(* IEC 61131-3 sources: IODBLib/, 7 files *)

(* ---- IODBLib.typ ---- *)
(********************************************************************
 * COPYRIGHT -- ARG
 ********************************************************************
 * Library: IODatabase
 * File: IODatabase.typ
 * Author: Administrator
 * Created: June 17, 2011
 ********************************************************************
 * Data types of library IODatabase
 ********************************************************************)

TYPE
	IODataBase : 	STRUCT
		Buffer : REFERENCE TO UDINT; (*Pointer to the allocated memory*)
		BufferSize : UDINT; (*size of the allocated memory*)
		DataTypeSize : UDINT; (*size of IODatapoint type*)
		ListDP : AsIOListDP; (*function block to get the IO on the system*)
		PVInfo : AsIOPVInfo; (*function block to get the PV's connected to the IO on the system*)
		State : USINT;
		NumberVariables : UINT;
	END_STRUCT;
	IODataPoint : 	STRUCT  (*DO NOT CHANGE ORDER: PVName, IODPType, INAName, IODPName*)
		PVName : STRING[80]; (*Name of the connected process variable*)
		IODPType : STRING[20]; (*Type of IO Point that is connected*)
		INAName : STRING[80]; (*INA address to slice*)
		IODPName : STRING[80]; (*Name of the connected IO datapoint*)
	END_STRUCT;
	Task_typ : 	STRUCT
		Name : STRING[80];
		Ident : UDINT;
		Group : USINT;
		State : USINT;
		Resource : SINT;
	END_STRUCT;
END_TYPE

(* ---- CreateIODatabase.st ---- *)
(********************************************************************
 * COPYRIGHT -- ARG
 ********************************************************************
 * Library: IODatabase
 * File: InitIODatabase.st
 * Author: Josh Polansky
 * Created: June 17, 2011
 ********************************************************************
 * Implementation of library IODatabase
 ********************************************************************)

//This MUST be called in INIT and must finish before calling GetINAInfo()

//Goes through all the IO and finds the number of connected datapoints

//Allocates memory

//Fills memory with datapoint info

FUNCTION CreateIODB

//Set return value to get rid of compiler warning

CreateIODB:=	0;

FOR iteration:= 0 TO 5 DO
	CASE Database.State OF

		1://Init
			Database.NumberVariables:=0;
			Database.ListDP.pLastDatapoint:= 0;
			Database.ListDP.enable:=1;
			Database.ListDP();
			IF Database.ListDP.status = 0 THEN
			  	Database.State:= 	2;
			END_IF

		2://We have a datapoint!
			IF Database.ListDP.pDatapoint <> 0
				THEN
			  	Database.State := 				3;
				Database.PVInfo.index:=			0;
				Database.PVInfo.pDatapoint:=	Database.ListDP.pDatapoint;
				Database.PVInfo.enable:=		1;
				Database.PVInfo();
				TempString ACCESS Database.PVInfo.pDatapoint;
			ELSE
			  	Database.State := 	0;
				CreateIODB:=		1;
			END_IF

		3://Get the status

			Database.PVInfo();

			IF Database.PVInfo.status = 0 //We have the info
				THEN
			  	Database.State := 	4;
			ELSIF Database.PVInfo.status = ERR_FUB_BUSY //We are getting the info
				THEN

			ELSE	//We couldn't get info, get the next one
			  	Database.State := 	5;
			END_IF

		4://Parse
			IF Database.PVInfo.pPvName <> 0 THEN

				//Get the current place in the buffer
				DataPoint  ACCESS (Database.Buffer + (Database.NumberVariables * Database.DataTypeSize));

				//Set the PV Name
				TempString ACCESS Database.PVInfo.pPvName;
				DataPoint.PVName:=	TempString;

				//Set the IO Datapoint name
				TempString ACCESS Database.ListDP.pDatapoint;
				DataPoint.IODPName:=	TempString;

				//Get the IO Type
				strind:=0;
				Done:=0;
				WHILE strind < brsstrlen(Database.ListDP.pDatapoint)
					AND strind < SIZEOF(DataPoint.IODPType)
					AND NOT Done
					DO
					IF	brsmemcmp( Database.ListDP.pDatapoint + strind,ADR('.'),1) = 0
					OR	brsmemcmp( Database.ListDP.pDatapoint + strind,ADR(':'),1) = 0
						THEN
						brsstrcpy( ADR(DataPoint.IODPType), Database.ListDP.pDatapoint );
						brsmemset( ADR(DataPoint.IODPType) + strind, 0, SIZEOF(DataPoint.IODPType)- strind);
						brsstrcpy( ADR(DataPoint.INAName),  Database.ListDP.pDatapoint + strind + 1 );
						Done:=1;
					END_IF
					strind:=strind+1;
				END_WHILE;

				len:= UDINT_TO_INT(brsstrlen( ADR(DataPoint.INAName) ));
				Done:=0;
				//Start at the end and look for the last "." to separate the INA device from the IODatapoint name
				WHILE( len > 0 AND NOT Done )  DO
					IF ( brsmemcmp( ADR(DataPoint.INAName) + len - 1, ADR('.' ), 1 ) = 0 )THEN
						Done := 1;
					END_IF
					TempString ACCESS ADR(DataPoint.INAName) + len - 1;
					len := len - 1;
				END_WHILE;

				brsstrcpy(ADR(DataPoint.IODPName),ADR(TempString)+1);
				TempString := '';

				Database.NumberVariables:= Database.NumberVariables+1;
				Database.State:= 	3;
				Database.PVInfo.index:=	Database.PVInfo.index+1;
			ELSE

				IF Database.PVInfo.index = 0 THEN
					Database.PVInfo.index:=	1;
					Database.State:= 	3;
				ELSE
					Database.State:= 	5;
				END_IF
			END_IF

		5://Get the next one
			Database.ListDP.pLastDatapoint:= Database.ListDP.pDatapoint;
			Database.ListDP();
			IF Database.ListDP.status = 0
				THEN
			  	Database.State:= 	2;
			ELSIF Database.ListDP.pDatapoint = 0 THEN
				Database.State := 	0;
			END_IF

	END_CASE;
END_FOR

END_FUNCTION

(* ---- GetChannelNum.st ---- *)
(********************************************************************
 * COPYRIGHT --
 ********************************************************************
 * Library: DPLookup
 * File: GetChannelNum.st
 * Author: Josh
 * Created: November 12, 2012
 ********************************************************************
 * Implementation of library DPLookup
 ********************************************************************)

(*  *)
FUNCTION GetChannelNum

	pDatapoint ACCESS GetINAInfo(DataBase,Datapoint,DPName);

	IF ADR(pDatapoint) <> 0 THEN
		DPName:=RIGHT(pDatapoint.IODPName,2);
		GetChannelNum := brsatoi( ADR(DPName));
	END_IF

END_FUNCTION

(* ---- GetINAInfo.st ---- *)
(********************************************************************
 * COPYRIGHT -- ARG
 ********************************************************************
 * Library: IODatabase
 * File: GetINAInfo.st
 * Author: Josh Polansky
 * Created: June 20, 2011
 ********************************************************************
 * Implementation of library IODatabase
 ********************************************************************)

FUNCTION GetINAInfo

(****************************************)
(* Check for invalid database 			*)
(****************************************)

IF( DataBase.Buffer = 0 )THEN

	GetINAInfo:=	0;
	INADeviceName:=	'Database not initialized';

	RETURN;

END_IF

(****************************************************************************)
(* Search through database for a PVName which matches the Datapoint input	*)
(****************************************************************************)

pDatapoint ACCESS (DataBase.Buffer + (DataBase.DataTypeSize * index) );

WHILE pDatapoint.PVName <> Datapoint AND index < DataBase.BufferSize/ DataBase.DataTypeSize DO

	pDatapoint ACCESS (DataBase.Buffer + (DataBase.DataTypeSize * index) );
	index:= index+1;

END_WHILE;

(****************************************)
(* Set return value						*)
(****************************************)

IF pDatapoint.PVName = Datapoint THEN

	GetINAInfo:=	ADR(pDatapoint);
	INADeviceName:=	pDatapoint.INAName;

ELSE

	GetINAInfo:=	0;
	INADeviceName:=	'Datapoint not found';

END_IF

END_FUNCTION

(* ---- InitIODatabase.st ---- *)
(*
 * File: InitIODatabase.st
 * Copyright (c) 2023 Loupe
 * https://loupe.team
 *
 * This file is part of IODBLib, licensed under the MIT License.
 *)

//This MUST be called in INIT and must finish before calling GetINAInfo()

//Goes through all the IO and finds the number of connected datapoints

//Allocates memory

//Fills memory with datapoint info

FUNCTION InitIODB

//Set return value to get rid of compiler warning

InitIODB:=	0;

//Get size of required buffer

Database.Buffer:=		0;
Database.BufferSize:=	0;
Database.DataTypeSize:=	SIZEOF( DataPoint);

//Get the first IO datapoint

Database.ListDP.pLastDatapoint:=	0;
Database.ListDP.enable:=			1;
Database.ListDP();

//Go through all the datapoints IO datapoints and check to see if they are connected to a PV datapoint

WHILE Database.ListDP.pDatapoint <> 0 // 0 means no datapoint was found
	DO

	Database.ListDP.pLastDatapoint:= Database.ListDP.pDatapoint;
	Database.ListDP();

	//If the status is 0 a datapoint was found

	IF ( Database.ListDP.status = 0 ) THEN

		//If we found a datapoint, check if it is connected to a PV

		Database.PVInfo.pDatapoint:=	Database.ListDP.pDatapoint;
		Database.PVInfo.enable:=		1;
		Database.PVInfo.index:=0;
		Database.PVInfo();
		IF Database.PVInfo.pDatapoint <> 0 THEN
			TempString ACCESS Database.PVInfo.pDatapoint;
//			logError('IOFound',TempString);
		END_IF

		//If there is a PV connected, add the size of the PV info to the buffer size

		//Get the producer
		IF Database.PVInfo.pPvName <> 0 THEN
			TempString ACCESS Database.PVInfo.pPvName;
//			logError('ProdPVFound',TempString);
			Database.BufferSize:= Database.BufferSize + Database.DataTypeSize;
		END_IF;

		Database.PVInfo.index:= Database.PVInfo.index+1;
		Database.PVInfo();

		//Get the Consumers
		WHILE Database.PVInfo.pPvName <> 0 DO
			TempString ACCESS Database.PVInfo.pPvName;
//			logError('ConsPVFound',TempString);
			Database.BufferSize:= Database.BufferSize + Database.DataTypeSize;
			Database.PVInfo.index:= Database.PVInfo.index+1;
			Database.PVInfo();
		END_WHILE;

	END_IF

END_WHILE;

//Get buffer

IF ( TMP_alloc(	Database.BufferSize,ADR(Database.Buffer)) = 0 )THEN
	Database.State:=1;
END_IF

END_FUNCTION

(* ---- GetTaskInfo.st ---- *)
(*
 * File: GetTaskInfo.st
 * Copyright (c) 2023 Loupe
 * https://loupe.team
 *
 * This file is part of IODBLib, licensed under the MIT License.
 *)

(*  *)
FUNCTION_BLOCK GetTaskInfo

	CASE State OF
		0:
			Status:= ERR_FUB_BUSY;
			IF ST_name(0,ADR(Info.Name),ADR(Info.Group)) = 0 THEN
				State:=1;
			END_IF

		1:
			IF ST_ident(ADR(Info.Name),Info.Group,ADR(Info.Ident)) = 0 THEN
				State:=2;
			END_IF

		2:
			IF ST_info(Info.Ident,ADR(Info.State),ADR(Info.Resource)) = 0 THEN
				Status:= ERR_OK;
				State:=3;
			END_IF

	END_CASE

END_FUNCTION_BLOCK

(* ---- IODBLib.fun ---- *)
(*
 * File: IODBLib.fun
 * Copyright (c) 2023 Loupe
 * https://loupe.team
 *
 * This file is part of IODBLib, licensed under the MIT License.
 *)

FUNCTION InitIODB : UINT
	VAR_INPUT
		Database : IODataBase;
	END_VAR
	VAR
		TempString : REFERENCE TO STRING[80];
		DataPoint : REFERENCE TO IODataPoint;
	END_VAR
END_FUNCTION

FUNCTION CreateIODB : USINT
	VAR_INPUT
		Database : IODataBase;
	END_VAR
	VAR
		TempString : REFERENCE TO STRING[80];
		DataPoint : REFERENCE TO IODataPoint;
		Done : BOOL;
		len : INT;
		strind : USINT;
		iteration : USINT;
	END_VAR
END_FUNCTION

FUNCTION GetINAInfo : UDINT
	VAR_INPUT
		DataBase : IODataBase;
		Datapoint : STRING[80];
	END_VAR
	VAR_IN_OUT
		INADeviceName : STRING[80];
	END_VAR
	VAR
		pDatapoint : REFERENCE TO IODataPoint;
		index : UINT;
	END_VAR
END_FUNCTION

FUNCTION GetChannelNum : DINT
	VAR_INPUT
		DataBase : IODataBase;
		Datapoint : STRING[80];
	END_VAR
	VAR
		pDatapoint : REFERENCE TO IODataPoint;
		DPName : STRING[80];
	END_VAR
END_FUNCTION

FUNCTION_BLOCK GetTaskInfo
	VAR_OUTPUT
		Info : Task_typ;
		Status : UINT;
	END_VAR
	VAR
		State : USINT;
	END_VAR
END_FUNCTION_BLOCK
